# B&R Automation Studio project POlaba1
Automation Studio 4.12.2.93

## Configuration Config1

CPU 4PP065.0571-P74, AutomationRuntime D4.52, Build 4.1.2, Vc V4.52.0

### Task classes (Cpu.sw)
```
Cyclic#1:
  Program <- Program.prg
Binaries: udbdef, TCData, ashwd, User, asfw, arconfig, sysconf, Role, ashwac, iomap
Libraries: MotContr
```

### Hardware
```
4PP065_0571_P74 : 4PP065.0571-P74 v1.1.2.0
  Connector IF4:
    DNAConfiguration = manual
  Connector IF5:
    ActivateDevice = 1
  ConfigurationID = POlaba1_Config1
  Simulation = 1
```

## Logical view

Binary libraries used (declarations not repeated): operator, runtime, astime, AsIecCon

### Library Logical/Libraries/MotContr (ANSIC)

#### MotContr.fun - Exported functions and function blocks
```iecst
{REDUND_ERROR} FUNCTION_BLOCK FB_Motor (*ДПТ*) (*$GROUP=User,$CAT=User,$GROUPICON=User.png,$CATICON=User.png*)
	VAR_INPUT
		u : REAL; (*Входное напряжение, В*)
		dt : REAL; (*Период дискретизации, с*)
	END_VAR
	VAR_OUTPUT
		w : REAL; (*Частота вращени, об./мин.*)
		phi : REAL; (*Положение вала, об.*)
	END_VAR
	VAR
		Tm : REAL; (*Механическая постоянная времени, с*)
		integrator : FB_Integrator; (*Интегратор*)
		ke : REAL; (*Постоянная ЭДС двигателя, В/(об./мин.)*)
	END_VAR
END_FUNCTION_BLOCK

{REDUND_ERROR} FUNCTION_BLOCK FB_Integrator (*Интегратор*) (*$GROUP=User,$CAT=User,$GROUPICON=User.png,$CATICON=User.png*)
	VAR_INPUT
		in : REAL; (*Вход*)
		dt : REAL; (*Период дискретизации, с*)
	END_VAR
	VAR_OUTPUT
		out : REAL; (*Выход*)
	END_VAR
	VAR
		prev_value : REAL; (*Предыдущее значение*)
	END_VAR
END_FUNCTION_BLOCK

{REDUND_ERROR} FUNCTION_BLOCK FB_Regulator (*ПИ-регулятор*) (*$GROUP=User,$CAT=User,$GROUPICON=User.png,$CATICON=User.png*)
	VAR_INPUT
		e_in : REAL; (*Вход (ошибка)*)
		dt : REAL; (*Период дискретизации, с*)
	END_VAR
	VAR_OUTPUT
		u_out : REAL; (*Выход*)
	END_VAR
	VAR
		k_p : REAL; (*Коэффициент пропорционального звена*)
		k_i : REAL; (*Коэффициент интегрального звена*)
		integrator : FB_Integrator; (*Интегратор*)
		iyOld : REAL; (*Предыдущее значение схемы противонакопления*)
		max_abs_value : REAL; (*Ограничение*)
		last_sum : REAL; (*Разница между предыдущими значениями u и sum*)
		sum : REAL; (*Выходное значение до звена ограничения*)
	END_VAR
END_FUNCTION_BLOCK
```

#### FB_Integrator.c
```c
#include <bur/plctypes.h>
#ifdef __cplusplus
	extern "C"
	{
#endif
	#include "MotContr.h"
#ifdef __cplusplus
	};
#endif
/* TODO: Add your comment here */
void FB_Integrator(struct FB_Integrator* inst)
{
	/*TODO: Add your code here*/
	inst->out = inst->dt * inst->in + inst->prev_value;
	inst->prev_value = inst->out;
}
```

#### FB_Regulator.c
```c
#include <bur/plctypes.h>
#ifdef __cplusplus
	extern "C"
	{
#endif
	#include "MotContr.h"
#ifdef __cplusplus
	};
#endif
/* TODO: Add your comment here */
void FB_Regulator(struct FB_Regulator* inst)
{
	inst->integrator.dt = inst->dt;

	REAL a = inst->e_in * inst->k_p;
	REAL b = inst->e_in * inst->k_i;

	a = a > inst->max_abs_value ? inst->max_abs_value : a;
	a = a < -inst->max_abs_value ? -inst->max_abs_value : a;

	inst->integrator.in = b + inst->last_sum;
	FB_Integrator(&inst->integrator);

	inst->sum = a + inst->integrator.out;
	inst->u_out = inst->sum;
	inst->u_out = inst->u_out > inst->max_abs_value ? inst->max_abs_value : inst->u_out;
	inst->u_out = inst->u_out < -inst->max_abs_value ? -inst->max_abs_value : inst->u_out;

	inst->last_sum = inst->u_out - inst->sum;
}
```

#### FB_Motor.c
```c
#include <bur/plctypes.h>
#ifdef __cplusplus
	extern "C"
	{
#endif
	#include "MotContr.h"
#ifdef __cplusplus
	};
#endif
/* TODO: Add your comment here */
void FB_Motor(struct FB_Motor* inst)
{
	inst->integrator.dt = inst->dt;
	REAL a = inst->u / inst->ke - inst->w;
	REAL b = a / inst->Tm;

	inst->integrator.in = b;
	FB_Integrator(&inst->integrator);

	inst->w = inst->integrator.out;
}
```

### Program Logical/Program

#### Variables.var
```iecst
VAR
	fb_controller : FB_Regulator;
	fb_motor1 : FB_Motor;
	fb_motor2 : FB_Motor;
	speed : REAL;
	counter : UINT;
	Tm : REAL;
	enable : BOOL;
	dt : REAL;
	u : REAL;
	ke : REAL;
END_VAR
```

#### Cyclic.c
```c
#include <bur/plctypes.h>

#ifdef _DEFAULT_INCLUDES
	#include <AsDefault.h>
#endif

void _CYCLIC ProgramCyclic(void)
{
	if(enable)
	{
		if(counter == 200)
		{
			speed = 50;
		}
		if(counter == 400)
		{
			speed = 0;
			counter = 0;
		}
		counter = counter + 1;

		fb_controller.e_in = speed - fb_motor1.w;
		FB_Regulator(&fb_controller);

		fb_motor1.u = fb_controller.u_out;
		FB_Motor(&fb_motor1);

		fb_motor2.u = speed * fb_motor2.ke;
		FB_Motor(&fb_motor2);
	}
}
```

#### Init.c
```c
#include <bur/plctypes.h>

#ifdef _DEFAULT_INCLUDES
	#include <AsDefault.h>
#endif

void _INIT ProgramInit(void)
{
	dt = 0.01;
	ke = 0.00265;
	Tm = 0.0246;
	u = 0;

	fb_motor1.dt = dt;
	fb_motor1.ke = ke;
	fb_motor1.Tm = Tm;
	fb_motor1.u = u;

	fb_motor2.dt = dt;
	fb_motor2.ke = ke;
	fb_motor2.Tm = Tm;
	fb_motor2.u = u;

	fb_controller.dt = dt;
	fb_controller.k_i = 0.053;
	fb_controller.k_p = 0.0013;
	fb_controller.max_abs_value = 24;

	speed = 0;
	counter = 0;
	enable = 1;
}
```

Listed in the project but not available here: Logical/Libraries/MotContr/Types.typ, Logical/Libraries/MotContr/Constants.var
